// TIA Portal V20 export
FUNCTION_BLOCK "LER_StackMainReady"   // FB96, LAD
// stored: Access Published, MemoryReserve 100, SetENOAutomatically false
   VAR_INPUT
      enable : Bool;
      reset : Bool;
      electrodeRemainValue : Bool;
      partData : Struct
         EM4 : "LER_typePartDataEm4";
         EM5 : "LER_typePartDataEm5";
         EM6 : "LER_typePartDataEm6";
         EM7 : "LER_typePartDataEm7";
         clearData : "LER_typePartData";
      END_STRUCT;
   END_VAR
   VAR_OUTPUT
      autoReady : Bool;
   END_VAR
BEGIN
END_FUNCTION_BLOCK
